{attribute 'enable_dynamic_creation'}
FUNCTION_BLOCK FB_SetDO EXTENDS FB_BaseAction
VAR
	// SetDO specific properties
	outputId : INT;
	value : BOOL;
END_VAR

// SetDO implementation

END_FUNCTION_BLOCK

(* stored: Version 1.1.0.1
   POU FB_SetDO: Id {f1b2c3d4-7775-7777-7777-777777777777} *)
